// TIA Portal V18 export
ORGANIZATION_BLOCK "19-Canopy"   // OB129, LAD, ProgramCycle
TITLE = "Main Program Sweep (Cycle)"
{ S7_Optimized_Access := 'TRUE' }
VERSION : 0.1
// stored: AutoNumber true, IsIECCheckEnabled false, SetENOAutomatically false
   VAR_INPUT
      Initial_Call : Bool;   // Initial call of this OB
      Remanence : Bool;   // =True, if remanent data are available
   END_VAR
   VAR_TEMP
      "Temp_1 (NormScale) Wire" : Real;
      "Temp_2 (NormScale) Inclanation" : Real;
      Temp_3 : Real;
      "Temp_4 (Radyan)" : Real;
      Temp_5 : Real;
      "Temp-6 AnimasyonNorm" : Real;
   END_VAR
   VAR_TEMP   // added for the SCL form of the ladder/FBD networks
      _w1 : Bool;
      _w2 : Bool;
      _w3 : Bool;
      _w4 : Bool;
      _w5 : Bool;
   END_VAR
BEGIN

REGION Network 1: Canopy
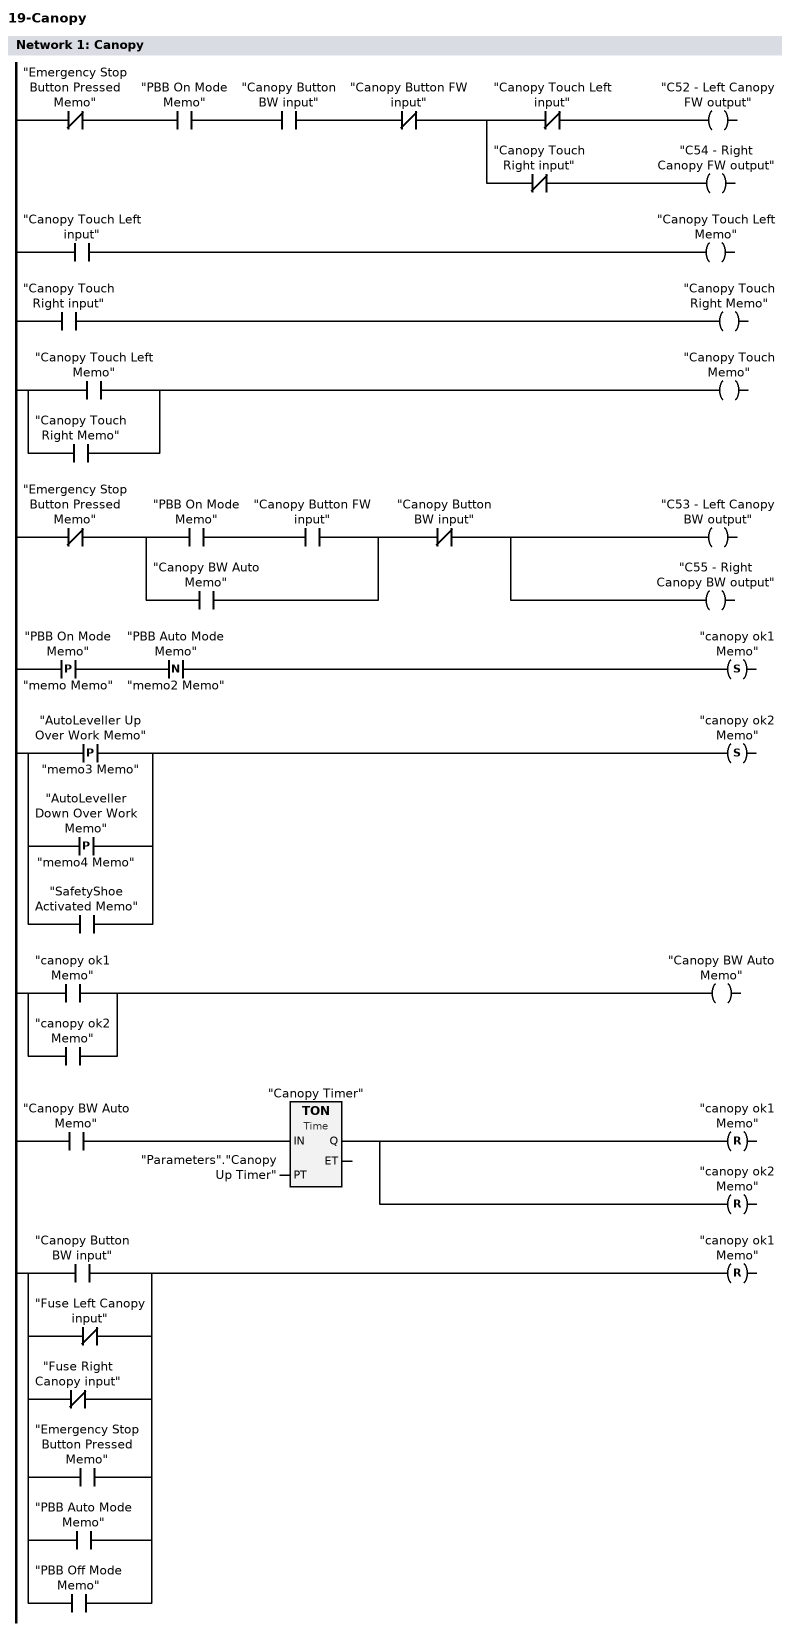
   RUNG wire#powerrail
      I_Contact( "Emergency Stop Button Pressed Memo" )
      Contact( "PBB On Mode Memo" )
      Contact( "Canopy Button BW input" )
      I_Contact( "Canopy Button FW input" )
      wire#w1
      I_Contact( "Canopy Touch Left input" )
      Coil( "C52 - Left Canopy FW output" )
   END_RUNG
   RUNG wire#w1
      I_Contact( "Canopy Touch Right input" )
      Coil( "C54 - Right Canopy FW output" )
   END_RUNG
   RUNG wire#powerrail
      Contact( "Canopy Touch Left input" )
      Coil( "Canopy Touch Left Memo" )
   END_RUNG
   RUNG wire#powerrail
      Contact( "Canopy Touch Right input" )
      Coil( "Canopy Touch Right Memo" )
   END_RUNG
   RUNG wire#powerrail
      Contact( "Canopy Touch Left Memo" )
      wire#w2
      Coil( "Canopy Touch Memo" )
   END_RUNG
   RUNG wire#powerrail
      Contact( "Canopy Touch Right Memo" )
   END_RUNG wire#w2
   RUNG wire#powerrail
      I_Contact( "Emergency Stop Button Pressed Memo" )
      wire#w3
      Contact( "PBB On Mode Memo" )
      Contact( "Canopy Button FW input" )
      wire#w4
      I_Contact( "Canopy Button BW input" )
      wire#w5
      Coil( "C53 - Left Canopy BW output" )
   END_RUNG
   RUNG wire#w3
      Contact( "Canopy BW Auto Memo" )
   END_RUNG wire#w4
   RUNG wire#w5
      Coil( "C55 - Right Canopy BW output" )
   END_RUNG
   RUNG wire#powerrail
      P_Contact(operand := "PBB On Mode Memo", bit := "memo Memo")
      N_Contact(operand := "PBB Auto Mode Memo", bit := "memo2 Memo")
      S_Coil( "canopy ok1 Memo" )
   END_RUNG
   RUNG wire#powerrail
      P_Contact(operand := "AutoLeveller Up Over Work Memo", bit := "memo3 Memo")
      wire#w6
      S_Coil( "canopy ok2 Memo" )
   END_RUNG
   RUNG wire#powerrail
      P_Contact(operand := "AutoLeveller Down Over Work Memo", bit := "memo4 Memo")
   END_RUNG wire#w6
   RUNG wire#powerrail
      Contact( "SafetyShoe Activated Memo" )
   END_RUNG wire#w6
   RUNG wire#powerrail
      Contact( "canopy ok1 Memo" )
      wire#w7
      Coil( "Canopy BW Auto Memo" )
   END_RUNG
   RUNG wire#powerrail
      Contact( "canopy ok2 Memo" )
   END_RUNG wire#w7
   RUNG wire#powerrail
      Contact( "Canopy BW Auto Memo" )
      { S7_Templates := "time_type := Time" } "Canopy Timer".TON(pt := "Parameters"."Canopy Up Timer", et =>)
      wire#w8
      R_Coil( "canopy ok1 Memo" )
   END_RUNG
   RUNG wire#w8
      R_Coil( "canopy ok2 Memo" )
   END_RUNG
   RUNG wire#powerrail
      Contact( "Canopy Button BW input" )
      wire#w9
      R_Coil( "canopy ok1 Memo" )
   END_RUNG
   RUNG wire#powerrail
      I_Contact( "Fuse Left Canopy input" )
   END_RUNG wire#w9
   RUNG wire#powerrail
      I_Contact( "Fuse Right Canopy input" )
   END_RUNG wire#w9
   RUNG wire#powerrail
      Contact( "Emergency Stop Button Pressed Memo" )
   END_RUNG wire#w9
   RUNG wire#powerrail
      Contact( "PBB Auto Mode Memo" )
   END_RUNG wire#w9
   RUNG wire#powerrail
      Contact( "PBB Off Mode Memo" )
   END_RUNG wire#w9
   // the same network as SCL:
   #_w1 := NOT "Emergency Stop Button Pressed Memo" AND "PBB On Mode Memo" AND "Canopy Button BW input" AND NOT "Canopy Button FW input";
   "C52 - Left Canopy FW output" := #_w1 AND NOT "Canopy Touch Left input";
   "C54 - Right Canopy FW output" := #_w1 AND NOT "Canopy Touch Right input";
   "Canopy Touch Left Memo" := "Canopy Touch Left input";
   "Canopy Touch Right Memo" := "Canopy Touch Right input";
   "Canopy Touch Memo" := "Canopy Touch Left Memo" OR "Canopy Touch Right Memo";
   "C53 - Left Canopy BW output" := NOT "Emergency Stop Button Pressed Memo" AND (("PBB On Mode Memo" AND "Canopy Button FW input") OR "Canopy BW Auto Memo") AND NOT "Canopy Button BW input";
   "C55 - Right Canopy BW output" := "C53 - Left Canopy BW output";
   #_w2 := "PBB On Mode Memo" AND NOT "memo Memo";   // rising edge of "PBB On Mode Memo"
   "memo Memo" := "PBB On Mode Memo";
   #_w3 := #_w2 AND NOT "PBB Auto Mode Memo" AND "memo2 Memo";   // falling edge of "PBB Auto Mode Memo"
   "memo2 Memo" := "PBB Auto Mode Memo";
   IF #_w3 THEN "canopy ok1 Memo" := TRUE; END_IF;
   #_w4 := "AutoLeveller Up Over Work Memo" AND NOT "memo3 Memo";   // rising edge of "AutoLeveller Up Over Work Memo"
   "memo3 Memo" := "AutoLeveller Up Over Work Memo";
   #_w5 := "AutoLeveller Down Over Work Memo" AND NOT "memo4 Memo";   // rising edge of "AutoLeveller Down Over Work Memo"
   "memo4 Memo" := "AutoLeveller Down Over Work Memo";
   IF #_w4 OR #_w5 OR "SafetyShoe Activated Memo" THEN "canopy ok2 Memo" := TRUE; END_IF;
   "Canopy BW Auto Memo" := "canopy ok1 Memo" OR "canopy ok2 Memo";
   "Canopy Timer".TON(IN := "Canopy BW Auto Memo", PT := "Parameters"."Canopy Up Timer");
   IF "Canopy Timer".Q THEN
       "canopy ok1 Memo" := FALSE;
       "canopy ok2 Memo" := FALSE;
   END_IF;
   IF "Canopy Button BW input" OR NOT "Fuse Left Canopy input" OR NOT "Fuse Right Canopy input" OR "Emergency Stop Button Pressed Memo" OR "PBB Auto Mode Memo" OR "PBB Off Mode Memo" THEN
       "canopy ok1 Memo" := FALSE;
   END_IF;
END_REGION
END_ORGANIZATION_BLOCK
